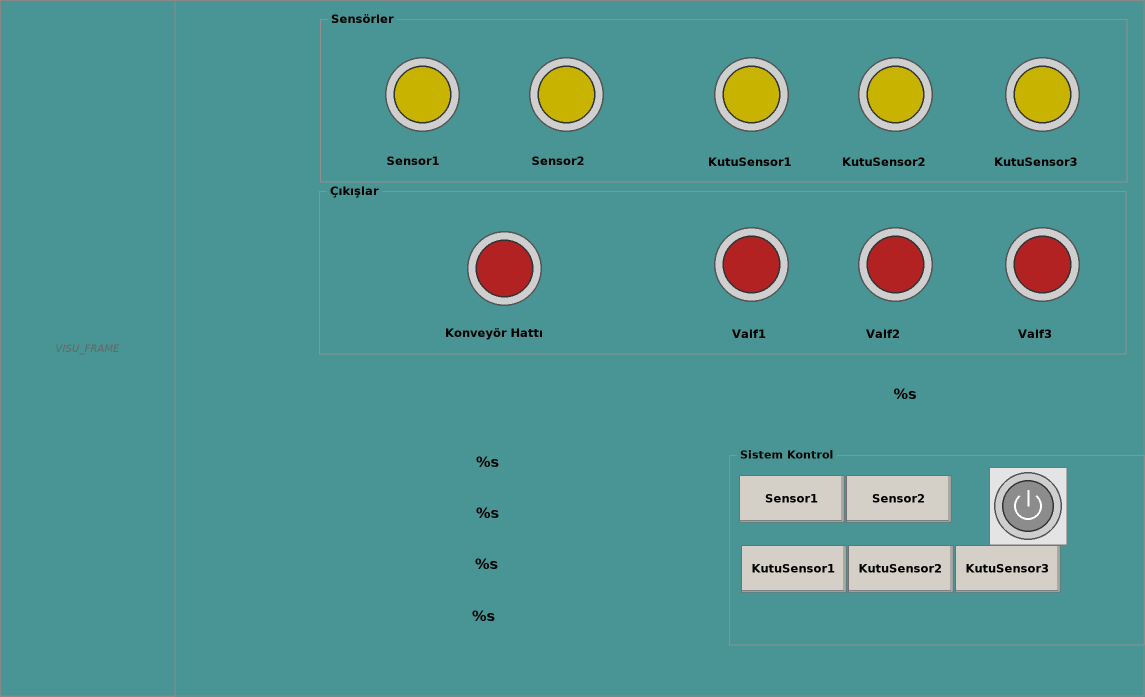
VISUALIZATION Visualization_1  // 1145x697
    Button (739,475 105x47), "Sensor1"
        toggle MAIN.bSensor1
    Button (846,475 105x47), "Sensor2"
        toggle MAIN.bSensor2
    Button (741,545 105x47), "KutuSensor1"
        toggle MAIN.bKutuSensor_1
    Button (848,545 105x47), "KutuSensor2"
        toggle MAIN.bKutuSensor_2
    Button (955,545 105x47), "KutuSensor3"
        toggle MAIN.bKutuSensor_3
    Lamp1 (370,51 105x87), variable: MAIN.bSensor1, style: Lamp-Lamp1-Yellow
    Lamp1 (514,51 105x87), variable: MAIN.bSensor2, style: Lamp-Lamp1-Yellow
    Lamp1 (699,51 105x87), variable: MAIN.bKutuSensor_1, style: Lamp-Lamp1-Yellow
    Lamp1 (843,51 105x87), variable: MAIN.bKutuSensor_2, style: Lamp-Lamp1-Yellow
    Lamp1 (990,51 105x87), variable: MAIN.bKutuSensor_3, style: Lamp-Lamp1-Yellow
    GroupBox (320,11 807x171), "Sensörler"
        Label (42,135 102x30), "Sensor1"
        Label (187,135 102x30), "Sensor2"
        Label (379,136 102x30), "KutuSensor1"
        Label (513,136 102x30), "KutuSensor2"
        Label (665,136 102x30), "KutuSensor3"
    Lamp1 (699,221 105x87), variable: MAIN.bValf1, style: Lamp-Lamp1-Red
    Lamp1 (843,221 105x87), variable: MAIN.bValf2, style: Lamp-Lamp1-Red
    Lamp1 (990,221 105x87), variable: MAIN.bValf3, style: Lamp-Lamp1-Red
    GroupBox (319,183 807x171), "Çıkışlar"
        Label (124,135 102x30), "Konveyör Hattı"
        Label (379,136 102x30), "Valf1"
        Label (513,136 102x30), "Valf2"
        Label (665,136 102x30), "Valf3"
        Lamp1 (133,42 105x87), variable: MAIN.bHat, style: Lamp-Lamp1-Red
    Rectangle (271,440 433x44), "%s", text variable: MAIN.sMsgInfo, text list: ''
    Rectangle (270,491 435x44), "%s", text variable: MAIN.sMsgKisa
    Rectangle (267,542 439x44), "%s", text variable: MAIN.sMsgOrta
    Rectangle (259,594 449x44), "%s", text variable: MAIN.sMsgUzun
    Rectangle (746,372 318x44), "%s", text variable: MAIN.sMsgMalzemeInfo
    Frame (0,0 175x697)
        shows VISU_FRAME(sDayTime := MAIN.DMY_LocalTime, sTime := MAIN.HMS_LocalTime)
    GroupBox (729,447 416x198), "Sistem Kontrol"
        PowerSwitch (257,20 84x78), variable: MAIN.bButton, behaviour: TOGGLE, style: Switch-PowerSwitch-Gray
END_VISUALIZATION

(* stored: Version 1.1.0.1, ProductVersion 3.1.4024.4
   Visu Visualization_1: Id {64ccad2f-747f-4c62-bc60-416b1b9ac1d1} *)
